Staubli VAL3: getMemoryFree.pgx

program getMemoryFree()
  local num l_nSpace
begin
  //
  l_nSpace=$getFreeSpace("/usr")
  gotoxy(1,9)
  put("sys free space:"+toString(".2",l_nSpace))
end
